// SIMATIC S7-200 SMART project (STEP 7-Micro/WIN SMART), CPU SR30

SYMBOL_TABLE 表格 1
停机fault          M2.0
报警fault          M2.1
中间变量3            M2.2
中间变量4            M2.3
中间变量5            M2.4
中间变量6            M2.5
中间变量7            M2.6
中间变量8            M2.7
中间变量9            M3.0
中间变量10           M3.1
中间变量11           M3.2
中间变量12           M3.3
中间变量13           M3.4
中间变量14           M3.5
中间变量15           M3.6
中间变量16           M3.7
液环泵手动1           V50.0
液环泵手动2           V50.1
入口阀手动1           V50.2
入口阀手动2           V50.3
补液阀手动            V50.4
排污阀手动            V50.5
调节阀手动            V50.6
液环泵1使能           V60.0
液环泵2使能           V60.1
入口阀1使能           V60.2
入口阀2使能           V60.3
液环泵fault1        V55.0
液环泵fault2        V55.1
流量开关fault        V55.2
急停fault          V55.3
温度报警fault        V55.4
温度停机fault        V55.5
低液位fault         V55.6
高液位fault         V55.7
真空值1             VD100
真空值2             VD104
温度值              VD108
液位值              VD112
低液位设定            VD116
高液位设定            VD120
目标液位             VD124
温度报警设定           VD128
温度急停设定           VD132
调节阀写入            VD136
系统真空值            VD140
目标真空             VD144
自动步骤             VW20
调节阀中间变量          VD148
调节阀手动参数          VD152
积分时间             VD156
微分时间             VD160
回路增益             VD164
END_SYMBOL_TABLE

SYMBOL_TABLE 系统符号
Always_On        SM0.0    // 始终接通
First_Scan_On    SM0.1    // 仅在第一个扫描周期时接通
Clock_1s         SM0.5    // 针对 1 s 的周期时间，时钟脉冲接通 0.5 s，断开 0.5 s.
END_SYMBOL_TABLE

ORGANIZATION_BLOCK MAIN:OB1
TITLE=程序注释
BEGIN
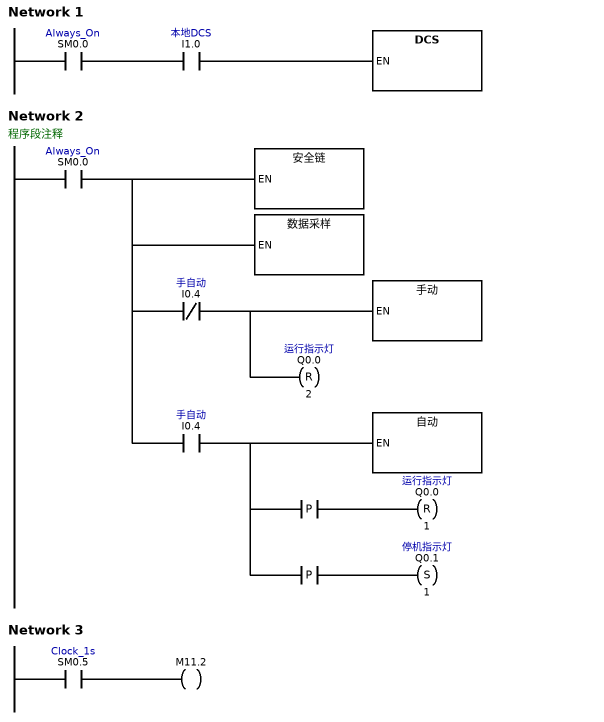
Network 1
LD     Always_On:SM0.0
A      本地DCS:I1.0
CALL   DCS:SBR2
Network 2
// 程序段注释
LD     Always_On:SM0.0
LPS
CALL   安全链:SBR3
CALL   数据采样:SBR4
AN     手自动:I0.4
CALL   手动:SBR0
R      运行指示灯:Q0.0, 2
LPP
A      手自动:I0.4
LPS
CALL   自动:SBR1
EU
R      运行指示灯:Q0.0, 1
LPP
EU
S      停机指示灯:Q0.1, 1
Network 3
LD     Clock_1s:SM0.5
=      M11.2
END_ORGANIZATION_BLOCK

SUBROUTINE_BLOCK 手动:SBR0
TITLE=子程序注释
BEGIN
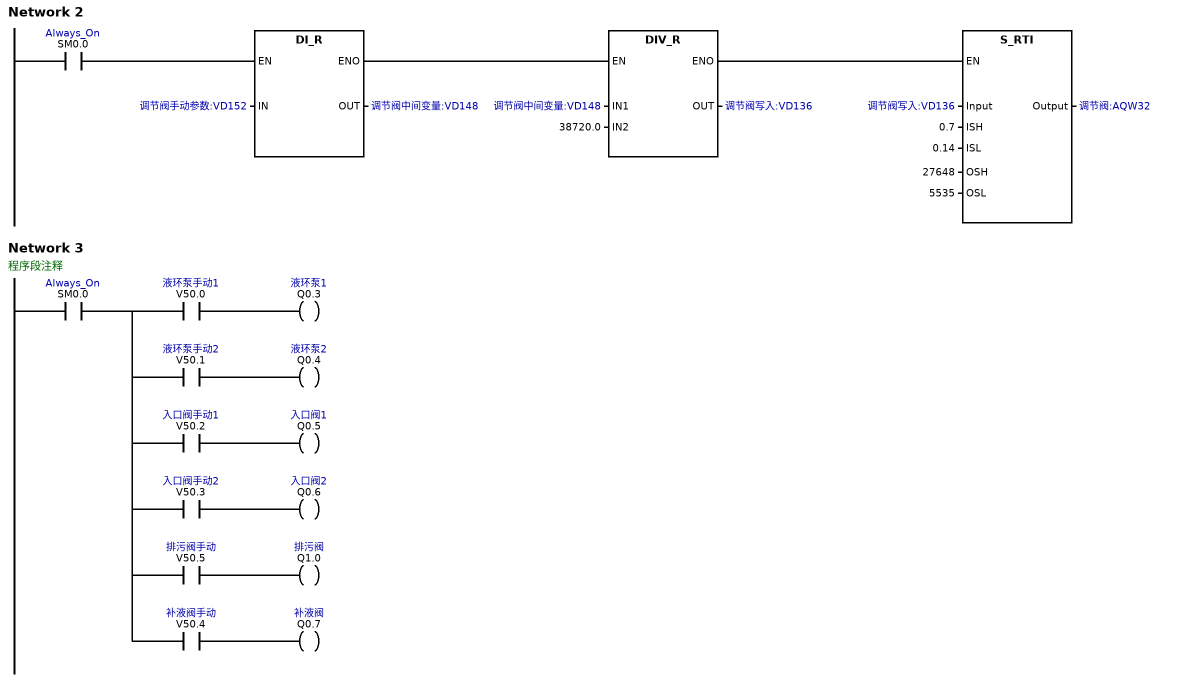
Network 2
LD     Always_On:SM0.0
DTR    调节阀手动参数:VD152, 调节阀中间变量:VD148
AENO
MOVR   调节阀中间变量:VD148, 调节阀写入:VD136
AENO
/R     38720.0, 调节阀写入:VD136
AENO
CALL   S_RTI:SBR5, 调节阀写入:VD136, 0.7, 0.14, 27648, 5535, 调节阀:AQW32
Network 3
// 程序段注释
LD     Always_On:SM0.0
LPS
A      液环泵手动1:V50.0
=      液环泵1:Q0.3
LRD
A      液环泵手动2:V50.1
=      液环泵2:Q0.4
LRD
A      入口阀手动1:V50.2
=      入口阀1:Q0.5
LRD
A      入口阀手动2:V50.3
=      入口阀2:Q0.6
LRD
A      排污阀手动:V50.5
=      排污阀:Q1.0
LPP
A      补液阀手动:V50.4
=      补液阀:Q0.7
END_SUBROUTINE_BLOCK

SUBROUTINE_BLOCK 自动:SBR1
TITLE=子程序注释
BEGIN
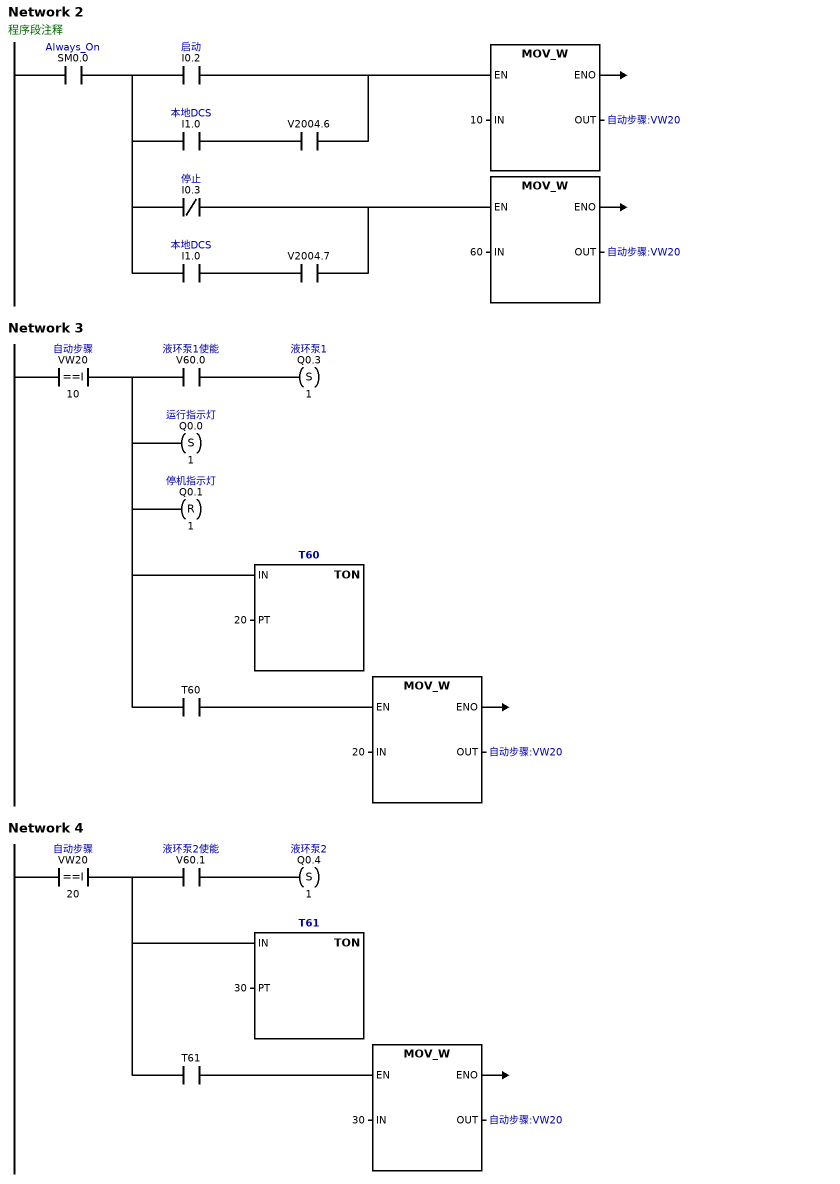
Network 2
// 程序段注释
LD     Always_On:SM0.0
LPS
LD     启动:I0.2
LD     本地DCS:I1.0
A      V2004.6
OLD
ALD
MOVW   10, 自动步骤:VW20
LPP
LDN    停止:I0.3
LD     本地DCS:I1.0
A      V2004.7
OLD
ALD
MOVW   60, 自动步骤:VW20
Network 3
LDW=   自动步骤:VW20, 10
LPS
A      液环泵1使能:V60.0
S      液环泵1:Q0.3, 1
LRD
S      运行指示灯:Q0.0, 1
LRD
R      停机指示灯:Q0.1, 1
LRD
TON    T60, 20
LPP
A      T60
MOVW   20, 自动步骤:VW20
Network 4
LDW=   自动步骤:VW20, 20
LPS
A      液环泵2使能:V60.1
S      液环泵2:Q0.4, 1
LRD
TON    T61, 30
LPP
A      T61
MOVW   30, 自动步骤:VW20
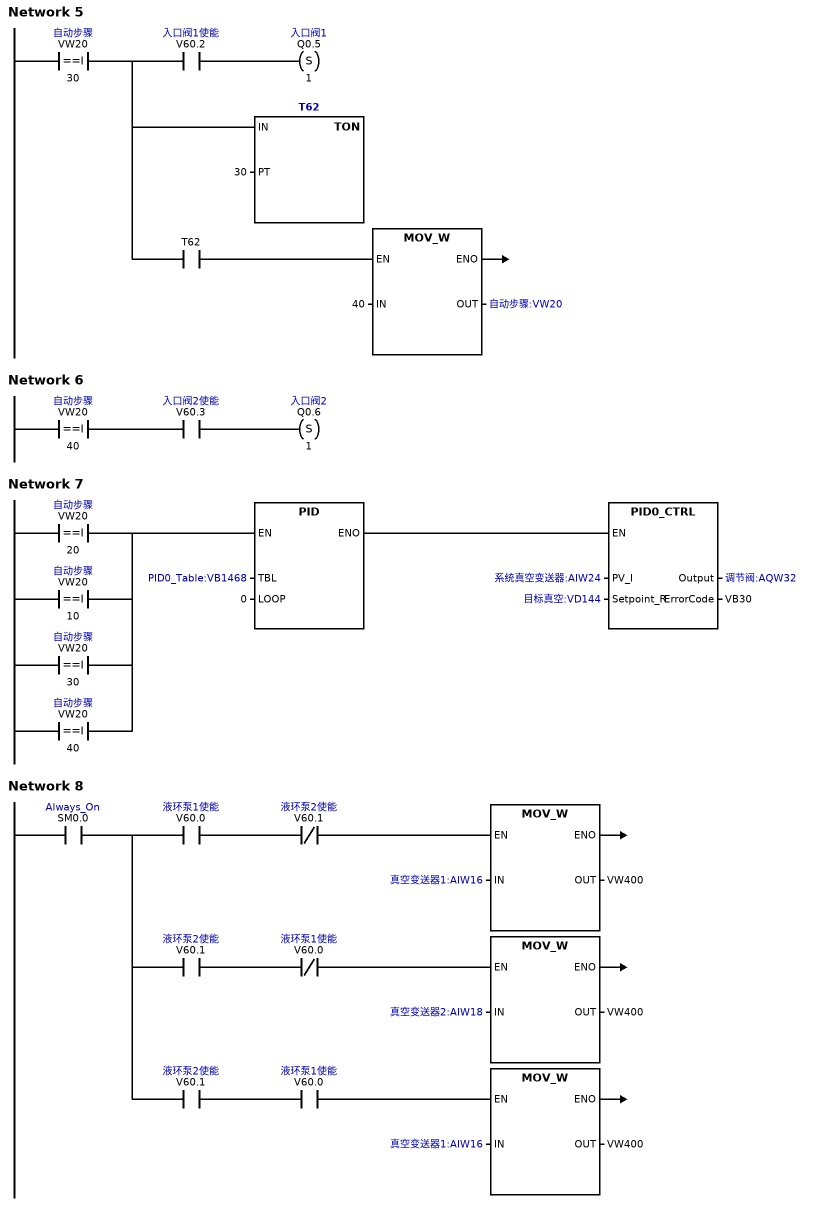
Network 5
LDW=   自动步骤:VW20, 30
LPS
A      入口阀1使能:V60.2
S      入口阀1:Q0.5, 1
LRD
TON    T62, 30
LPP
A      T62
MOVW   40, 自动步骤:VW20
Network 6
LDW=   自动步骤:VW20, 40
A      入口阀2使能:V60.3
S      入口阀2:Q0.6, 1
Network 7
LDW=   自动步骤:VW20, 20
OW=    自动步骤:VW20, 10
OW=    自动步骤:VW20, 30
OW=    自动步骤:VW20, 40
PID    PID0_Table:VB1468, 0
AENO
CALL   PID0_CTRL:SBR8, 系统真空变送器:AIW24, 目标真空:VD144, 调节阀:AQW32, VB30
Network 8
LD     Always_On:SM0.0
LPS
A      液环泵1使能:V60.0
AN     液环泵2使能:V60.1
MOVW   真空变送器1:AIW16, VW400
LRD
A      液环泵2使能:V60.1
AN     液环泵1使能:V60.0
MOVW   真空变送器2:AIW18, VW400
LPP
A      液环泵2使能:V60.1
A      液环泵1使能:V60.0
MOVW   真空变送器1:AIW16, VW400
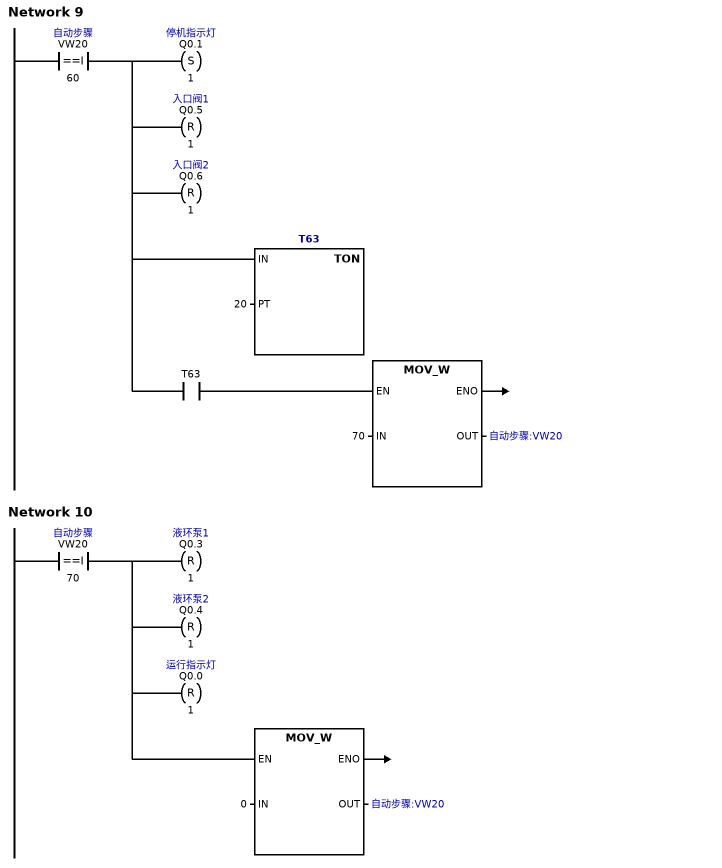
Network 9
LDW=   自动步骤:VW20, 60
S      停机指示灯:Q0.1, 1
R      入口阀1:Q0.5, 1
R      入口阀2:Q0.6, 1
TON    T63, 20
A      T63
MOVW   70, 自动步骤:VW20
Network 10
LDW=   自动步骤:VW20, 70
R      液环泵1:Q0.3, 1
R      液环泵2:Q0.4, 1
R      运行指示灯:Q0.0, 1
MOVW   0, 自动步骤:VW20
END_SUBROUTINE_BLOCK

SUBROUTINE_BLOCK DCS:SBR2
TITLE=子程序注释
BEGIN
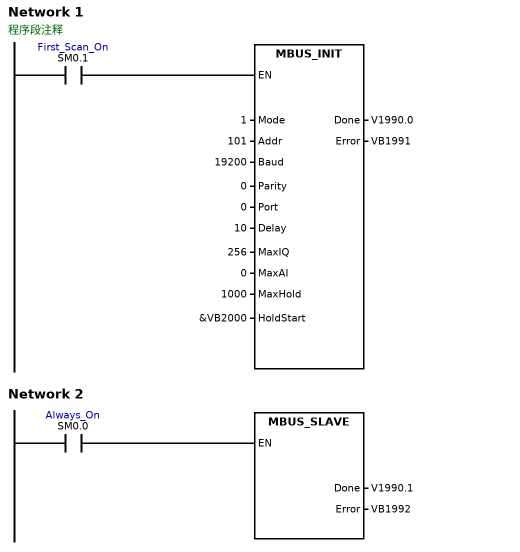
Network 1
// 程序段注释
LD     First_Scan_On:SM0.1
CALL   MBUS_INIT:SBR6, 1, 101, 19200, 0, 0, 10, 256, 0, 1000, &VB2000, V1990.0, VB1991
Network 2
LD     Always_On:SM0.0
CALL   MBUS_SLAVE:SBR9, V1990.1, VB1992
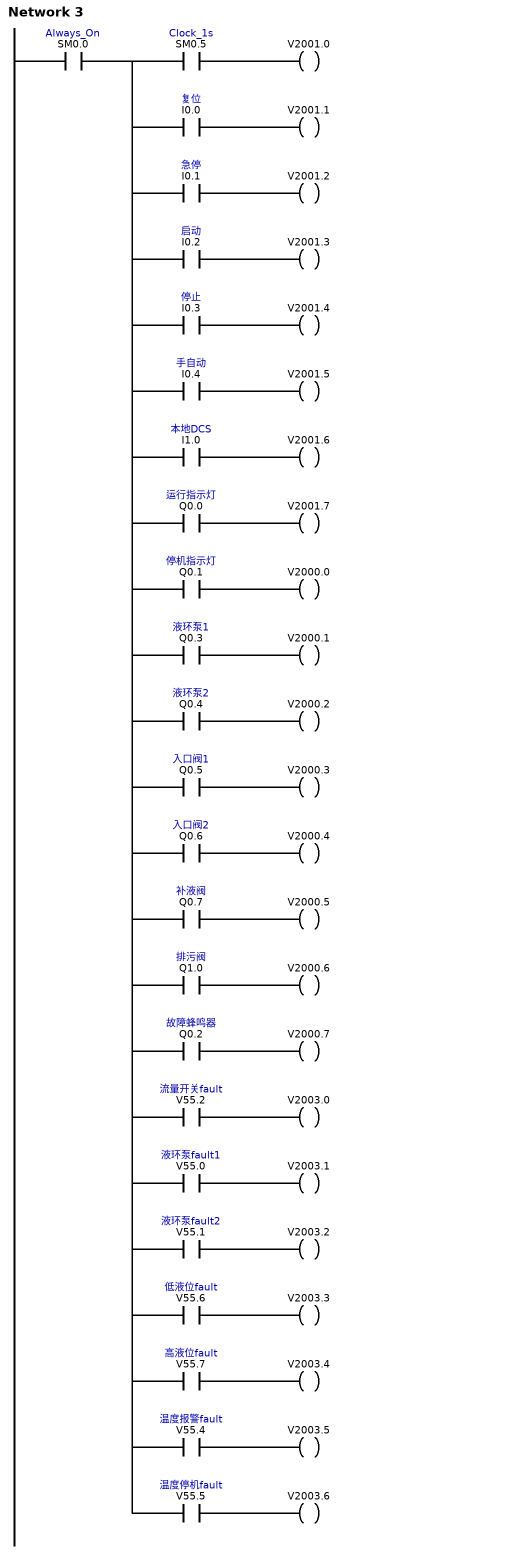
Network 3
LD     Always_On:SM0.0
LPS
A      Clock_1s:SM0.5
=      V2001.0
LRD
A      复位:I0.0
=      V2001.1
LRD
A      急停:I0.1
=      V2001.2
LRD
A      启动:I0.2
=      V2001.3
LRD
A      停止:I0.3
=      V2001.4
LRD
A      手自动:I0.4
=      V2001.5
LRD
A      本地DCS:I1.0
=      V2001.6
LRD
A      运行指示灯:Q0.0
=      V2001.7
LRD
A      停机指示灯:Q0.1
=      V2000.0
LRD
A      液环泵1:Q0.3
=      V2000.1
LRD
A      液环泵2:Q0.4
=      V2000.2
LRD
A      入口阀1:Q0.5
=      V2000.3
LRD
A      入口阀2:Q0.6
=      V2000.4
LRD
A      补液阀:Q0.7
=      V2000.5
LRD
A      排污阀:Q1.0
=      V2000.6
LRD
A      故障蜂鸣器:Q0.2
=      V2000.7
LRD
A      流量开关fault:V55.2
=      V2003.0
LRD
A      液环泵fault1:V55.0
=      V2003.1
LRD
A      液环泵fault2:V55.1
=      V2003.2
LRD
A      低液位fault:V55.6
=      V2003.3
LRD
A      高液位fault:V55.7
=      V2003.4
LRD
A      温度报警fault:V55.4
=      V2003.5
LPP
A      温度停机fault:V55.5
=      V2003.6
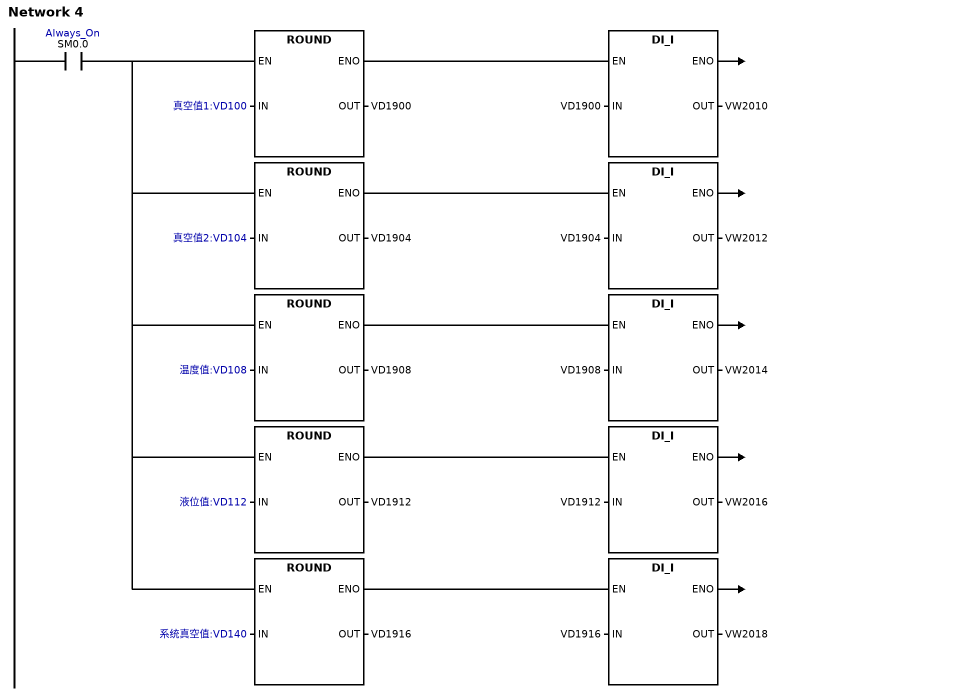
Network 4
LD     Always_On:SM0.0
LPS
ROUND  真空值1:VD100, VD1900
AENO
DTI    VD1900, VW2010
LRD
ROUND  真空值2:VD104, VD1904
AENO
DTI    VD1904, VW2012
LRD
ROUND  温度值:VD108, VD1908
AENO
DTI    VD1908, VW2014
LRD
ROUND  液位值:VD112, VD1912
AENO
DTI    VD1912, VW2016
LPP
ROUND  系统真空值:VD140, VD1916
AENO
DTI    VD1916, VW2018
END_SUBROUTINE_BLOCK

SUBROUTINE_BLOCK 安全链:SBR3
TITLE=子程序注释
BEGIN
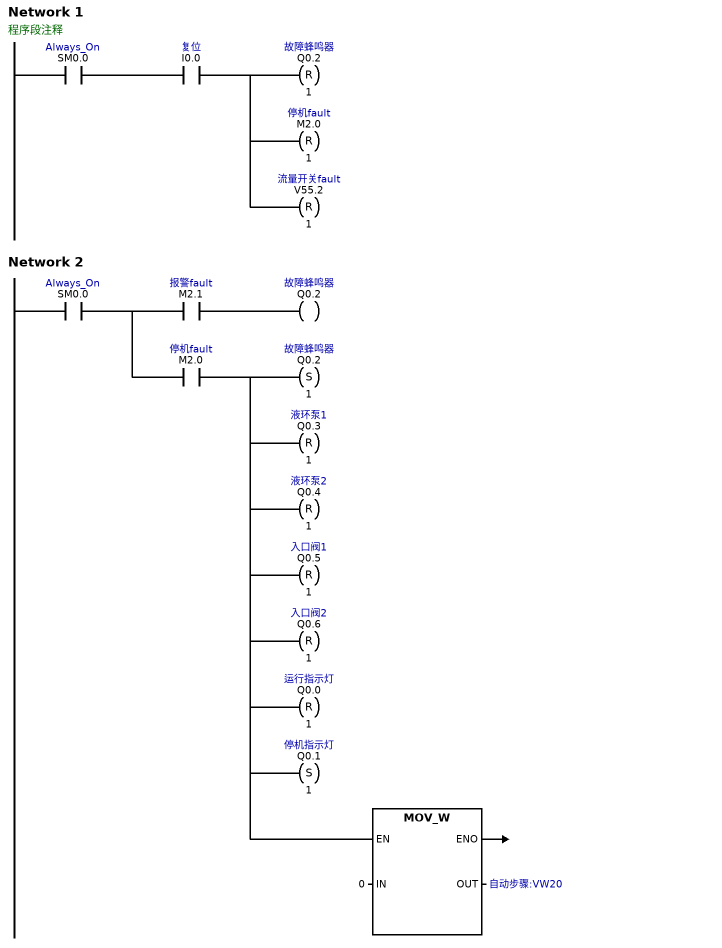
Network 1
// 程序段注释
LD     Always_On:SM0.0
A      复位:I0.0
R      故障蜂鸣器:Q0.2, 1
R      停机fault:M2.0, 1
R      流量开关fault:V55.2, 1
Network 2
LD     Always_On:SM0.0
LPS
A      报警fault:M2.1
=      故障蜂鸣器:Q0.2
LPP
A      停机fault:M2.0
S      故障蜂鸣器:Q0.2, 1
R      液环泵1:Q0.3, 1
R      液环泵2:Q0.4, 1
R      入口阀1:Q0.5, 1
R      入口阀2:Q0.6, 1
R      运行指示灯:Q0.0, 1
S      停机指示灯:Q0.1, 1
MOVW   0, 自动步骤:VW20
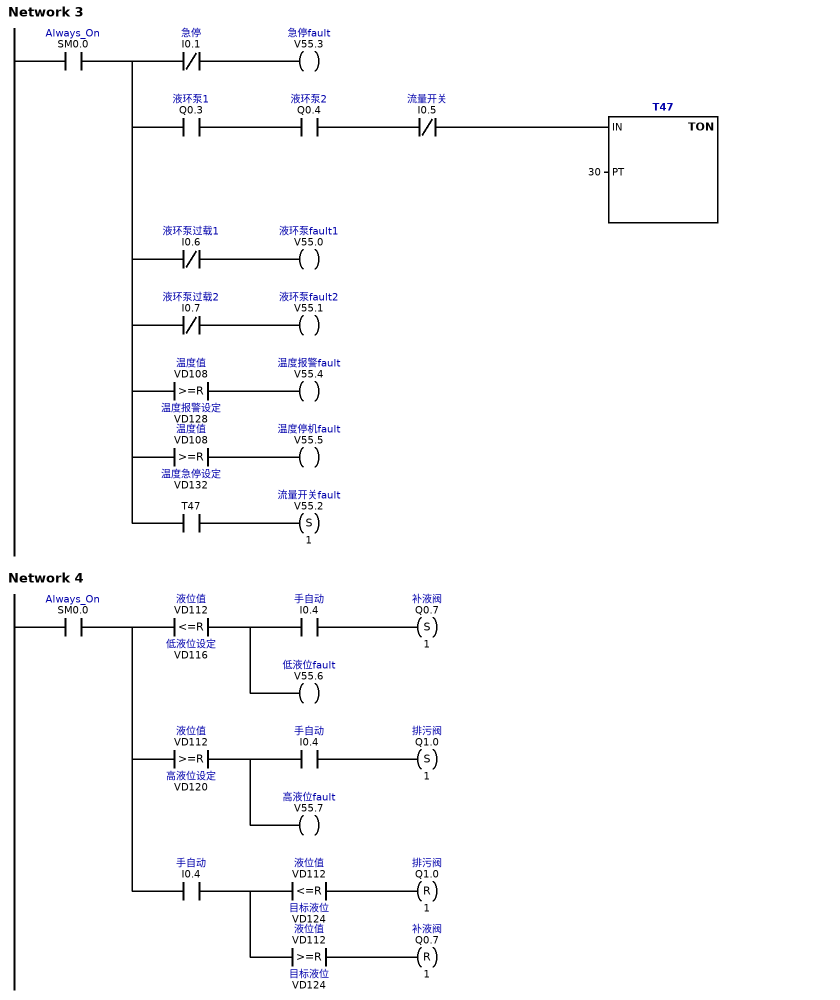
Network 3
LD     Always_On:SM0.0
LPS
AN     急停:I0.1
=      急停fault:V55.3
LRD
A      液环泵1:Q0.3
A      液环泵2:Q0.4
AN     流量开关:I0.5
TON    T47, 30
LRD
AN     液环泵过载1:I0.6
=      液环泵fault1:V55.0
LRD
AN     液环泵过载2:I0.7
=      液环泵fault2:V55.1
LRD
AR>=   温度值:VD108, 温度报警设定:VD128
=      温度报警fault:V55.4
LRD
AR>=   温度值:VD108, 温度急停设定:VD132
=      温度停机fault:V55.5
LPP
A      T47
S      流量开关fault:V55.2, 1
Network 4
LD     Always_On:SM0.0
LPS
AR<=   液位值:VD112, 低液位设定:VD116
LPS
A      手自动:I0.4
S      补液阀:Q0.7, 1
LPP
=      低液位fault:V55.6
LRD
AR>=   液位值:VD112, 高液位设定:VD120
LPS
A      手自动:I0.4
S      排污阀:Q1.0, 1
LPP
=      高液位fault:V55.7
LPP
A      手自动:I0.4
LPS
AR<=   液位值:VD112, 目标液位:VD124
R      排污阀:Q1.0, 1
LPP
AR>=   液位值:VD112, 目标液位:VD124
R      补液阀:Q0.7, 1
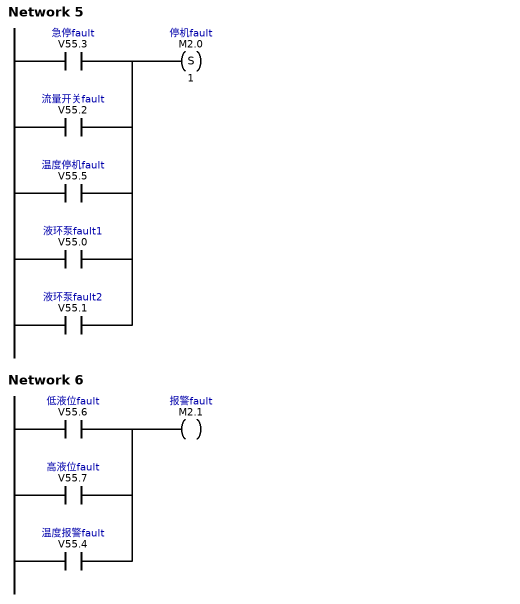
Network 5
LD     急停fault:V55.3
O      流量开关fault:V55.2
O      温度停机fault:V55.5
O      液环泵fault1:V55.0
O      液环泵fault2:V55.1
S      停机fault:M2.0, 1
Network 6
LD     低液位fault:V55.6
O      高液位fault:V55.7
O      温度报警fault:V55.4
=      报警fault:M2.1
END_SUBROUTINE_BLOCK

SUBROUTINE_BLOCK 数据采样:SBR4
TITLE=子程序注释
BEGIN
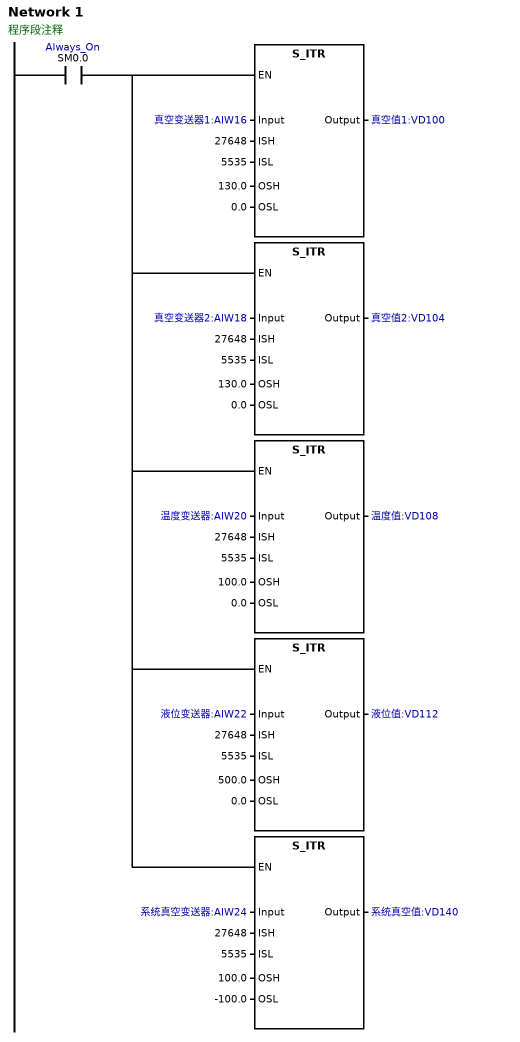
Network 1
// 程序段注释
LD     Always_On:SM0.0
CALL   S_ITR:SBR7, 真空变送器1:AIW16, 27648, 5535, 130.0, 0.0, 真空值1:VD100
CALL   S_ITR:SBR7, 真空变送器2:AIW18, 27648, 5535, 130.0, 0.0, 真空值2:VD104
CALL   S_ITR:SBR7, 温度变送器:AIW20, 27648, 5535, 100.0, 0.0, 温度值:VD108
CALL   S_ITR:SBR7, 液位变送器:AIW22, 27648, 5535, 500.0, 0.0, 液位值:VD112
CALL   S_ITR:SBR7, 系统真空变送器:AIW24, 27648, 5535, 100.0, -100.0, 系统真空值:VD140
END_SUBROUTINE_BLOCK

// SBR5: protected block, not included

// SBR6: protected block, not included

// SBR7: protected block, not included

// SBR8: protected block, not included

// SBR9: protected block, not included

// SBR10: protected block, not included

// INT1: protected block, not included
